FUNCTION_BLOCK EG_a2 (* Basic FB with empty ECC *)
  (* Standard: 61499-2 *)
  (* Version 1.0, 0000-00-00, 0 *)
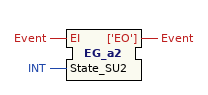
  EVENT_INPUT
    EI;
  END_EVENT
  EVENT_OUTPUT
    ['EO'];
  END_EVENT
  VAR_INPUT
    State_SU2 : INT;
  END_VAR
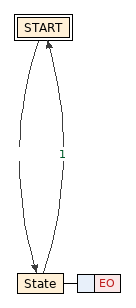
  EC_STATES
    START; (* Initial State *)
    State : -> EO;
  END_STATES
  EC_TRANSITIONS
    START TO State := ;
    State TO START := 1;
  END_TRANSITIONS
END_FUNCTION_BLOCK
(* other elements stored in the file *)
(* With Var=State_SU2 *)
